(* IEC 61131-3 sources: eCockpitGit/test_project/src/%F%00 Library/%F%Common Functions/%F%Filter, 1 file *)

(* ---- %POU%FB_diSampleFilter.st ---- *)
FUNCTION_BLOCK FB_diSampleFilter
VAR_OUTPUT
	currentValue		:DINT;
	amountSamples		:BYTE;
END_VAR
VAR
	samples				:POINTER TO ARRAY[0..255] OF DINT;
	position			:BYTE;
END_VAR
(*%!%__DELIMITER__%!%*)
